PROGRAM MAIN
VAR
END_VAR

Motion();

//PrgMqttCom();

END_PROGRAM

(* stored: Version 1.1.0.1, ProductVersion 3.1.4024.12
   POU MAIN: Id {7b2dc756-732b-421e-93a7-bb1631fbf9b8}, SpecialFunc None *)
